(* CODESYS project FU_sConcat10.xml

Project tree, tasks and I/O mapping:
  function FU_sConcat10 [ST]
*)

// FU_sConcat10
//This functions combines ten strings
// |**Version**|**Author**| **Date** |**Changes**
// | 1         | NSN      | 03-12-18 | Creation
FUNCTION FU_sConcat10 : STRING(255)
VAR_INPUT
	s1			:STRING(255);			//Input String1
	s2			:STRING(255);			//Input String2
	s3			:STRING(255);			//Input String3
	s4			:STRING(255);			//Input String4
	s5			:STRING(255);			//Input String5
	s6			:STRING(255);			//Input String6
	s7			:STRING(255);			//Input String7
	s8			:STRING(255);			//Input String8
	s9			:STRING(255);			//Input String9
	s10			:STRING(255);			//Input String10
END_VAR

FU_sConcat10BIBO(sOut:=ADR(FU_sConcat10),s1:=ADR(s1),s2:=ADR(s2),s3:=ADR(s3),s4:=ADR(s4),s5:=ADR(s5),s6:=ADR(s6),s7:=ADR(s7),s8:=ADR(s8),s9:=ADR(s9),s10:=ADR(s10),wOutSize:=255);

END_FUNCTION
